INTERFACE I_XP_Enviroment_PLC EXTENDS I_CH_Object

{attribute 'monitoring':='call'}
(* If Enable, the movers are checked for collisions with each other.
Warning and error can have their own size offsets.
The error leads to a stop with higher dynamics.
In simulation, an error does not lead to a stop *)
PROPERTY CollisionCheck : BOOL
GET
END_GET
SET
END_SET
END_PROPERTY

{attribute 'monitoring':='call'}
//Offset on the mover dimension from the MC3 mover object [mm] ;
// >0 menas the warning is earlier
PROPERTY MoverCollisionOffsetError : LREAL
GET
END_GET
SET
END_SET
END_PROPERTY

{attribute 'monitoring':='call'}
//Offset on the mover dimension from the MC3 mover object [mm] ;
// >0 menas the warning is earlier
PROPERTY MoverCollisionOffsetWarning : LREAL
GET
END_GET
SET
END_SET
END_PROPERTY

{attribute 'monitoring':='call'}
//Enumeration MoverDetectionStatus
PROPERTY MoverDetectionStatus : MoverDetectionStatus
GET
END_GET
END_PROPERTY

{attribute 'monitoring':='call'}
//Object ID of the IoXPlanar processing unit
PROPERTY ProcessingUnitOID : OTCID
GET
END_GET
END_PROPERTY

{attribute 'monitoring':='call'}
//Interface to CHALET system to which this object belongs
PROPERTY System : I_XP_System_PLC
GET
END_GET
END_PROPERTY

END_INTERFACE

(* stored: Version 1.1.0.1, ProductVersion 3.1.4024.13
   Itf I_XP_Enviroment_PLC: Id {d23b004d-987a-48e1-9bb8-d66144d5420d}
   Property CollisionCheck: Id {183e7718-bb80-4fa3-a30c-dcc44c977a72}
   Get Get: Id {a4b3e746-8b58-4f3f-b279-0929739e7062}
   Set Set: Id {f3e1d737-e39d-4738-80e6-b68b517f4fb9}
   Property MoverCollisionOffsetError: Id {438afaa6-2caa-4577-be67-f6a5f6345288}
   Get Get: Id {557ac927-4318-4085-9c57-546f4cc42b10}
   Set Set: Id {86de3990-3feb-423d-9c94-66d5157d305a}
   Property MoverCollisionOffsetWarning: Id {c214b6eb-65a6-4d1a-b4dc-e498f2a4177d}
   Get Get: Id {f21538ee-93fd-48ec-81bf-09a38400e38d}
   Set Set: Id {67d876f5-369e-48e8-95fe-ddaea6392db1}
   Property MoverDetectionStatus: Id {988a9ea0-160b-41bc-a976-d65943ed072c}
   Get Get: Id {fcca43c5-55b2-4a6f-9805-c64d279791fe}
   Property ProcessingUnitOID: Id {dd050f23-dd75-4380-abd4-9f9e80bf4ab2}
   Get Get: Id {f1baa752-a470-47d8-936f-8d777d44a21c}
   Property System: Id {64ddc72a-12e5-40c0-b185-6159ffa98088}
   Get Get: Id {5ec636f5-9a36-488a-9c13-85aa482137f4} *)
